{attribute 'GeneratedUsingTerminal: EL2212-0000-0018'}
{attribute addProperty BoxType "EL2212-0000-0018"}
{attribute addProperty Id "EtcSlaveTerminalBaseDOX_Status_Channel_1AT %I*DOX_Status_Channel_09DD45C87DOX_Status_Channel_2AT %I*DOX_Status_Channel_09DD45C87DOX_Control_Channel_1AT %Q*DOX_Control_Channel_A74F23633DOX_Control_Channel_2AT %Q*DOX_Control_Channel_A74F23633WcStateAT %I*WcState_9091E0EB2InfoDataAT %I*InfoData_32EB74EA10"}
{attribute addProperty CRC "1298761096"}
{attribute addProperty Size "32"}
TYPE EL2212_4D698588 EXTENDS EtcSlaveTerminalBase :
STRUCT
	{attribute addProperty Name "DOX_Status_Channel_1"}
	DOX_Status_Channel_1 : DOX_Status_Channel_09DD45C8;
	{attribute addProperty Name "DOX_Status_Channel_2"}
	DOX_Status_Channel_2 : DOX_Status_Channel_09DD45C8;
	{attribute addProperty Name "DOX_Control_Channel_1"}
	DOX_Control_Channel_1 : DOX_Control_Channel_A74F2363;
	{attribute addProperty Name "DOX_Control_Channel_2"}
	DOX_Control_Channel_2 : DOX_Control_Channel_A74F2363;
	{attribute addProperty Name "WcState"}
	WcState : WcState_9091E0EB;
	{attribute addProperty Name "InfoData"}
	InfoData : InfoData_32EB74EA;
END_STRUCT
END_TYPE

(* stored: Version 1.2.0.0, ProductVersion 3.1.4024.9
   DUT EL2212_4D698588: Id {afd8a225-769e-4c38-bb61-334119b91a30} *)
